(* CoDeSys 2.3 export: NETVAROD_SERVICE_UDP.EXP *)

(* Data type *)
TYPE NetVarOD_Service_Udp :
(
	ODStateFree := 0,
	ODReadRequest,
	ODReadRequestReply,
	ODWriteRequest,
	ODWriteRequestReply,
	ODAcknowledgement,
	ODBootUpRequest,

	ODErrorReplyUnnown := 20,
	ODErrorReplyItems,
	ODErrorReplyAccess,
	ODErrorReplyIdx,
	ODErrorReplySub,
	ODErrorReplyLen,

	ODErrorWrongService,
	ODErrorTimeOut,
	ODErrorReplyCPUStopped,

	ODStateBusy := 100
);
END_TYPE
